(* Logix 5000 project; controller Simulated_IO Emulate 5570 rev 36.11; software revision 36.00 *)

TASK MainTask (continuous, watchdog 500 ms) : MainProgram

MODULES
   Local : Emulate 5570 (ICP 2, rev 36.11)
      Simulat_IO : vendor 1 type 0 code 15 (ICP 3, rev 1.1, Output RPI 50 ms)
END_MODULES

ADD_ON_INSTRUCTION CONVEYOR   (* revision 1.0, vendor 2WRTECH *)
// Subcribe
// Help:
// Here is the description
VAR_INPUT
   LOC : BOOL; {access Read Only, required}
   REM : BOOL; {access Read Only, required}
   STRT : BOOL; {access Read Only, required}
   STOP : BOOL; {access Read Only, required}
   ESD : BOOL; {access Read Only, required}
   JOG : BOOL; {access Read Only, required}
END_VAR
VAR_OUTPUT
   RDY : BOOL; {visible}
   RUN : BOOL; {access Read Only, required}
   FB : BOOL; {access Read Only, required}
END_VAR
VAR_INPUT
   OL : BOOL; {access Read Only, required}
   TOL : BOOL; {access Read Only, required}
   CBK_TRIP : BOOL; {access Read Only, required}
END_VAR
VAR_OUTPUT
   FLT : BOOL; {access Read Only, visible}
   RUN_CMD : BOOL; {access Read Only}
END_VAR
VAR_INPUT
   RUN_DLY : DINT; {required}
   SPD_DLY : DINT; {required}
   RP_SW : BOOL; {required}
   DF_SW : BOOL; {required}
   SPD_SW : BOOL; {required}
   RST : BOOL; {required}
   RUN_SEC : DINT; {visible}
END_VAR
VAR_OUTPUT
   ALM_ROPE : BOOL; {access Read Only, visible}
   ALM_DRIFT : BOOL; {visible}
   ALM_ESD : BOOL; {access Read Only, visible}
   ALM_LOAD : BOOL; {access Read Only, visible}
   FB_LOSS : BOOL; {access Read Only, visible}
   BK_TRIP : BOOL; {access Read Only, visible}
   ALM_THERM : BOOL; {access Read Only, visible}
   ALM_SPEED : BOOL; {visible}
END_VAR
VAR
   STRT_DLY : TIMER := (PRE := 6000); {access None}
   SPEED_SW_DLY : TIMER := (PRE := 2000); {access None}
   PLC_DATE_TIME : DINT[7];
        [0]   // YEAR
        [1]   // MONTH
        [2]   // DAY
        [3]   // HOURS
        [4]   // MINUTE
        [6]   // MILLISECONDE
   OLD_SEC : DINT; {access None}
   PUL_SEC : BOOL[32]; {access None}
END_VAR

ROUTINE Logic   (* ladder *)
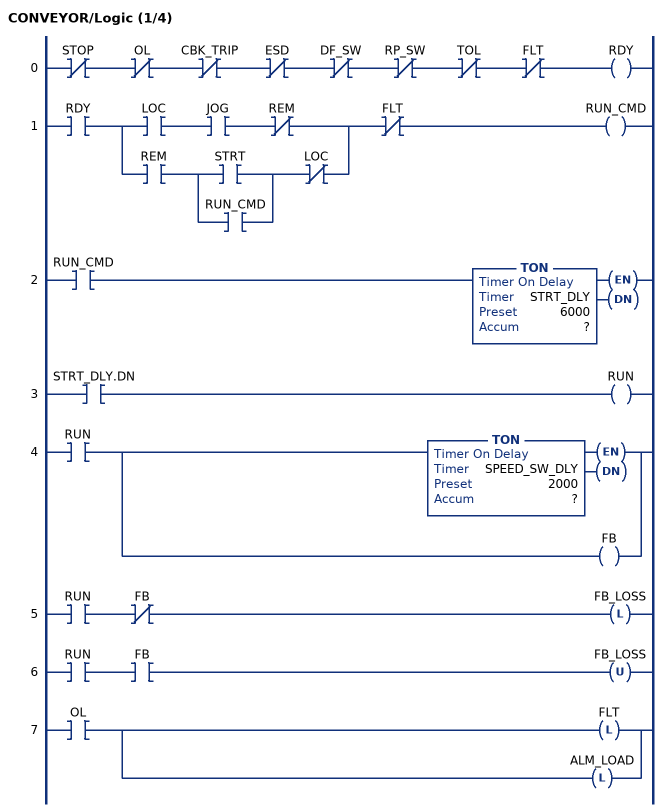
   0: XIO(STOP)XIO(OL)XIO(CBK_TRIP)XIO(ESD)XIO(DF_SW)XIO(RP_SW)XIO(TOL)XIO(FLT)OTE(RDY);
   1: XIC(RDY)[XIC(LOC) XIC(JOG) XIO(REM) ,XIC(REM) [XIC(STRT) ,XIC(RUN_CMD) ] XIO(LOC) ]XIO(FLT)OTE(RUN_CMD);
   2: XIC(RUN_CMD)TON(STRT_DLY,?,?);
   3: XIC(STRT_DLY.DN)OTE(RUN);
   4: XIC(RUN)[TON(SPEED_SW_DLY,?,?) ,OTE(FB) ];
   5: XIC(RUN)XIO(FB)OTL(FB_LOSS);
   6: XIC(RUN)XIC(FB)OTU(FB_LOSS);
   7: XIC(OL)[OTL(FLT) ,OTL(ALM_LOAD) ];
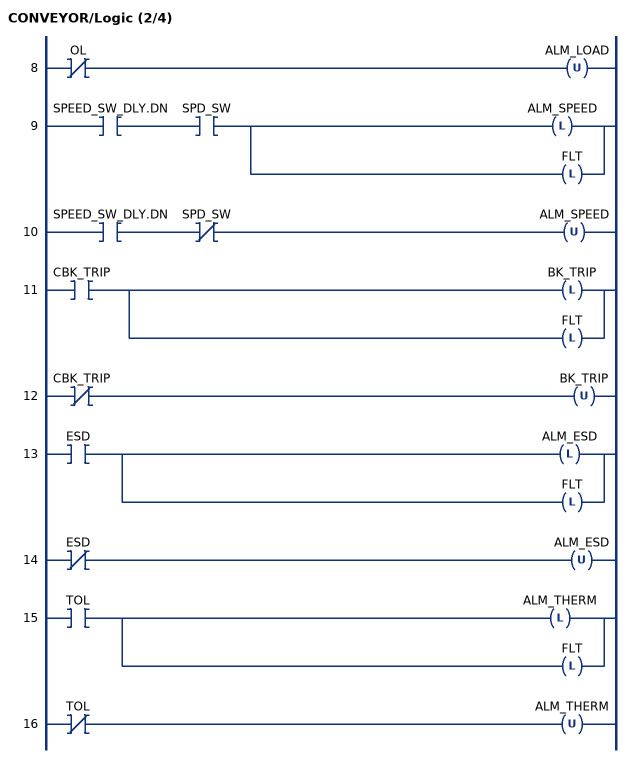
   8: XIO(OL)OTU(ALM_LOAD);
   9: XIC(SPEED_SW_DLY.DN)XIC(SPD_SW)[OTL(ALM_SPEED) ,OTL(FLT) ];
   10: XIC(SPEED_SW_DLY.DN)XIO(SPD_SW)OTU(ALM_SPEED);
   11: XIC(CBK_TRIP)[OTL(BK_TRIP) ,OTL(FLT) ];
   12: XIO(CBK_TRIP)OTU(BK_TRIP);
   13: XIC(ESD)[OTL(ALM_ESD) ,OTL(FLT) ];
   14: XIO(ESD)OTU(ALM_ESD);
   15: XIC(TOL)[OTL(ALM_THERM) ,OTL(FLT) ];
   16: XIO(TOL)OTU(ALM_THERM);
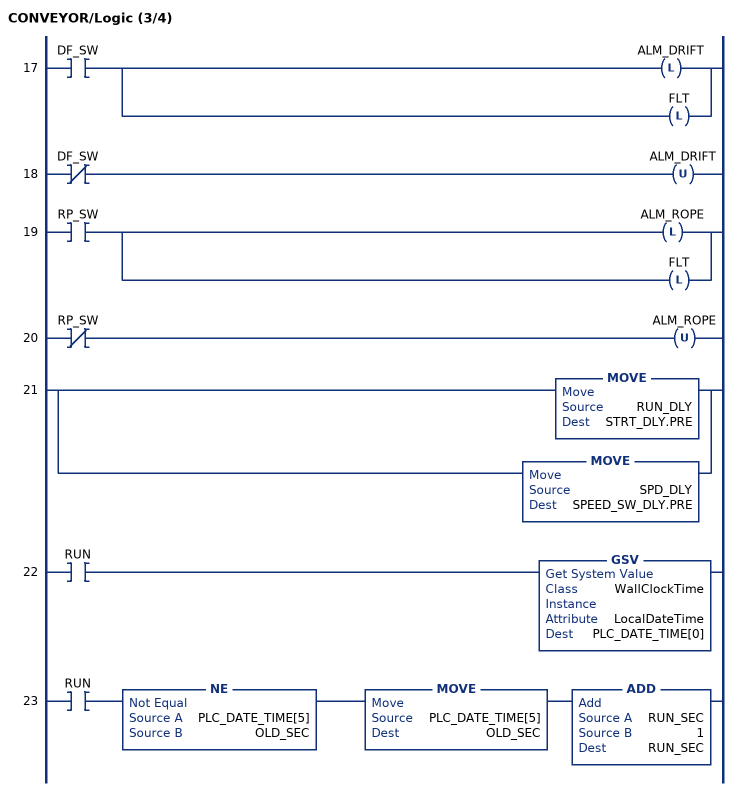
   17: XIC(DF_SW)[OTL(ALM_DRIFT) ,OTL(FLT) ];
   18: XIO(DF_SW)OTU(ALM_DRIFT);
   19: XIC(RP_SW)[OTL(ALM_ROPE) ,OTL(FLT) ];
   20: XIO(RP_SW)OTU(ALM_ROPE);
   21: [MOVE(RUN_DLY,STRT_DLY.PRE) ,MOVE(SPD_DLY,SPEED_SW_DLY.PRE) ];
   22: XIC(RUN)GSV(WallClockTime,,LocalDateTime,PLC_DATE_TIME[0]);
   23: XIC(RUN)NE(PLC_DATE_TIME[5],OLD_SEC)MOVE(PLC_DATE_TIME[5],OLD_SEC)ADD(RUN_SEC,1,RUN_SEC);
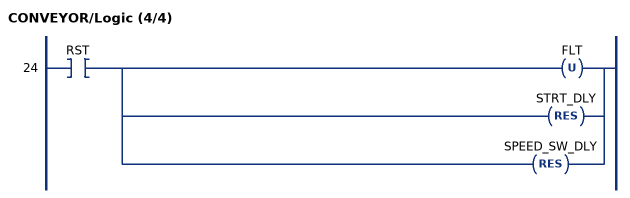
   24: XIC(RST)[OTU(FLT) ,RES(STRT_DLY) ,RES(SPEED_SW_DLY) ];
END_ROUTINE
END_ADD_ON_INSTRUCTION

VAR_GLOBAL   (* controller tags *)
   BELT_CONV : CONVEYOR;
   DRIFT_SW : BOOL;
   E_STOP : BOOL;
   FAULTED : BOOL;
   FB_RUN : BOOL;
   JOGGING : BOOL;
   LOCAL : BOOL;
   Output_En : BOOL;
   OVERLOAD : BOOL;
   REMOTE : BOOL;
   RESET : BOOL;
   ROPE_SW : BOOL;
   Speed_Delay : DINT;
   SPEED_SW : BOOL;
   Start_Delay : DINT;
   START_PB : BOOL;
   STOP_PB : BOOL;
   THERM : BOOL;
   TRIPPED : BOOL;
END_VAR

PROGRAM MainProgram   (* main routine MainRoutine *)

ROUTINE MainRoutine   (* ladder *)
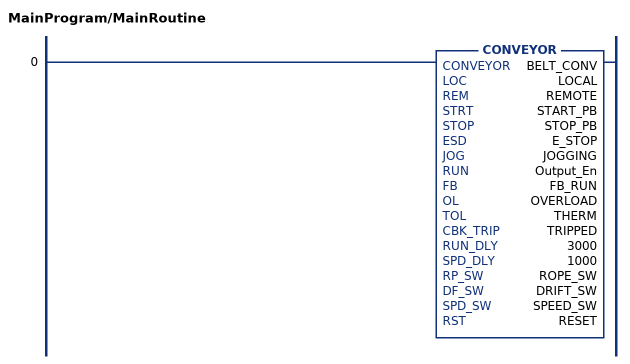
   0: CONVEYOR(BELT_CONV,LOCAL,REMOTE,START_PB,STOP_PB,E_STOP,JOGGING,Output_En,FB_RUN,OVERLOAD,THERM,TRIPPED,3000,1000,ROPE_SW,DRIFT_SW,SPEED_SW,RESET);
END_ROUTINE
END_PROGRAM
